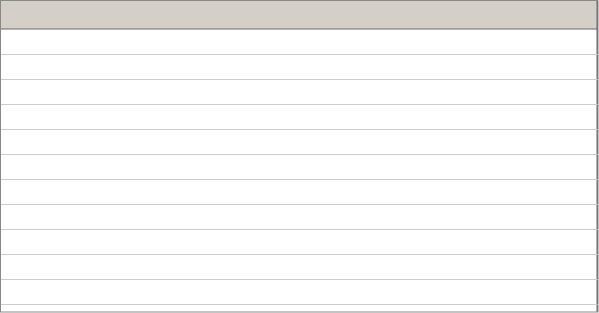
VISUALIZATION history  // 599x313
    Table (-2,-1 599x313), data array: AlarmManager.event_table_view.stAlarmhistory
        p3854506369: AlarmManager.event_table_view.stAlarmhistory[INDEX].nSourceId
        p1892666644: AlarmManager.event_table_view.stAlarmhistory[INDEX].nEventId
        p338671338: AlarmManager.event_table_view.stAlarmhistory[INDEX].Severity
        p2170511999: AlarmManager.event_table_view.stAlarmhistory[INDEX].ConfirmState
        p3723444502: AlarmManager.event_table_view.stAlarmhistory[INDEX].sDate
        p1218418051: AlarmManager.event_table_view.stAlarmhistory[INDEX].sTime
        p746581629: AlarmManager.event_table_view.stAlarmhistory[INDEX].Computer
        p3104783080: AlarmManager.event_table_view.stAlarmhistory[INDEX].sSource
        p2501879983: AlarmManager.event_table_view.stAlarmhistory[INDEX].MessageText
        p7306298: AlarmManager.event_table_view.stAlarmhistory[INDEX].bQuitMessage
        p1933151965: AlarmManager.event_table_view.stAlarmhistory[INDEX].bConfirmable
        p1755163831: 重要度
        p4092479075: 履歴
        p2237128397: 日付
        p505689113: 時刻
        p2243050616: テキスト
END_VISUALIZATION

(* stored: Version 1.1.0.1, ProductVersion 3.1.4024.15
   Visu history: Id {907c409e-ffbf-4347-b449-114ba4c76525} *)
